INTERFACE I_Status

PROPERTY Busy : BOOL
GET
END_GET
END_PROPERTY

PROPERTY Done : BOOL
GET
END_GET
END_PROPERTY

PROPERTY Error : BOOL
GET
END_GET
END_PROPERTY

PROPERTY ErrorID : UDINT
GET
END_GET
END_PROPERTY

PROPERTY Message : T_MAXSTRING
GET
END_GET
END_PROPERTY

END_INTERFACE

(* stored: Version 1.1.0.1
   Itf I_Status: Id {e55c9db0-e9ca-4cc5-89eb-efe222512305}
   Property Busy: Id {e5c844a7-f57a-4992-8e6c-c18ee2305d4c}
   Get Get: Id {c3eff79f-24e9-45f8-8ad9-0620eedd8e77}
   Property Done: Id {0f73ccbb-ed5a-4875-be60-9a747dc36d16}
   Get Get: Id {b4de3bc9-d738-4a49-affc-5024ca961374}
   Property Error: Id {efdc98a9-deec-47f6-8da6-128ddfab571a}
   Get Get: Id {827d2d58-2a69-4236-92f9-dd0f289ed438}
   Property ErrorID: Id {e6c661db-0a97-4c9d-92a6-213065012b2c}
   Get Get: Id {70f914e1-4cbc-49c1-b320-2ba7dbe224ec}
   Property Message: Id {bee1a366-8f68-49ab-be45-fcd4a5b3e66f}
   Get Get: Id {e045c474-98ea-48cc-97c6-72fa82ca43f1} *)
